(* CODESYS project introToSFC.export

Project tree, tasks and I/O mapping:
  Device : CODESYS Control Win V3 x64, CODESYS, version 3.5.22.30
    application Application
      libraries: Standard, 3.5.22.0 (System)
      task MainTask (cyclic, interval t#20ms, priority 1) calls PLC_PRG
      program PLC_PRG [SFC]
      program PLC_PRG_ST [ST]
*)

// Device/Application/PLC_PRG
PROGRAM PLC_PRG
VAR
	A: BOOL;
	B: BOOL;
	C: BOOL;
	Trans0A: BOOL;
	Trans0B: BOOL;
	Trans1: BOOL;
	Trans2: BOOL;
END_VAR

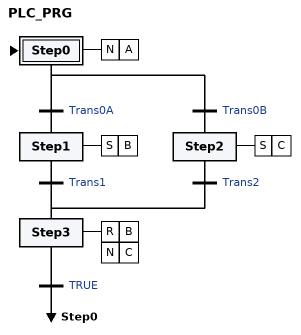
INITIAL_STEP Step0:
    A(N);
END_STEP
TRANSITION FROM Step0 TO Step1
    := Trans0A;
END_TRANSITION
STEP Step1:
    B(S);
END_STEP
TRANSITION FROM Step1 TO Step3
    := Trans1;
END_TRANSITION
TRANSITION FROM Step0 TO Step2
    := Trans0B;
END_TRANSITION
STEP Step2:
    C(S);
END_STEP
TRANSITION FROM Step2 TO Step3
    := Trans2;
END_TRANSITION
STEP Step3:
    B(R);
    C(N);
END_STEP
TRANSITION FROM Step3 TO Step0
    := TRUE;
END_TRANSITION

END_PROGRAM

// Device/Application/PLC_PRG_ST
PROGRAM PLC_PRG_ST
VAR
	A: BOOL;
	B: BOOL;
	C: BOOL;
	state: INT:=0;
	Trans0A: BOOL;
	Trans0B: BOOL;
	Trans1: BOOL;
	Trans2: BOOL;
END_VAR

CASE state OF
	//step0
	0:
	A:= TRUE;
	IF Trans0A THEN
		A:=FALSE;
		ELSIF Trans0B THEN
			A:=FALSE;
			state:=2;
	END_IF
	
	//step1
	1:
	B:=TRUE;
	IF Trans1 THEN
		state:=3;
	END_IF
	
	
	//step2
	2:
	C:=TRUE;
	IF Trans2 THEN
		state:=3;
	END_IF
	
	//step3
	3:
	B:=FALSE;
	C:=FALSE;
	state:=0;
END_CASE

END_PROGRAM
